// TIA Portal V16 export
// export: Created 2021-08-10T09:04:59.4784454Z, ExportSetting WithDefaults, WithReadOnly, DisplayName Totally Integrated Automation Portal, DisplayVersion V16, DisplayName TIA Portal Version Control Interface, DisplayVersion V16, DisplayName TIA Portal Openness, DisplayVersion V16, DisplayName TIA Portal Teamcenter Gateway, DisplayVersion V16, DisplayName SINAMICS Startdrive Advanced, DisplayVersion V16, DisplayName SINAMICS Startdrive G130, G150, S120, S150, SINAMICS MV, S210, DisplayVersion V16, DisplayName SINAMICS Startdrive G110M, G120, G120C, G120D, G120P, DisplayVersion V16, DisplayName STEP 7 Professional, DisplayVersion V16, DisplayName STEP 7 Safety, DisplayVersion V16, DisplayName WinCC Unified SCADA Engineering System, DisplayVersion V16
FUNCTION_BLOCK "Valve Liquid 2"   // FB3, FBD
{ S7_Optimized_Access := 'TRUE' }
VERSION : 0.1
// stored: AutoNumber true, CodeModifiedDate 2020-02-26T13:09:02.1361563Z, CompileDate 2021-07-03T08:38:43.4120873Z, CreationDate 2020-02-26T07:16:44.3135253Z, DownloadWithoutReinit false, HandleErrorsWithinBlock false, InterfaceModifiedDate 2020-02-26T12:49:56.0619358Z, IsConsistent true, IsIECCheckEnabled false, IsKnowHowProtected false, ISMultiInstanceCapable true, IsRetainMemResEnabled false, IsWriteProtected false, LibraryConformanceStatus Warning: The object contains access to global data blocks. Warning: The block contains direct access to inputs, outputs, bit memories, indirect access to the registry or indirect access to external memory areas that are unknown at the time of compilation., MemoryReserve 100, ModifiedDate 2020-02-26T13:09:02.1361563Z, ParameterModified 2020-02-26T07:16:44.3135253Z, PLCSimAdvancedSupport true, SetENOAutomatically false, StructureModified 2020-02-26T12:49:56.0619358Z, UDAEnableTagReadback false
   VAR
      VlvLiq2 : "fbValve_Solenoid";
   END_VAR
BEGIN

REGION Network 1
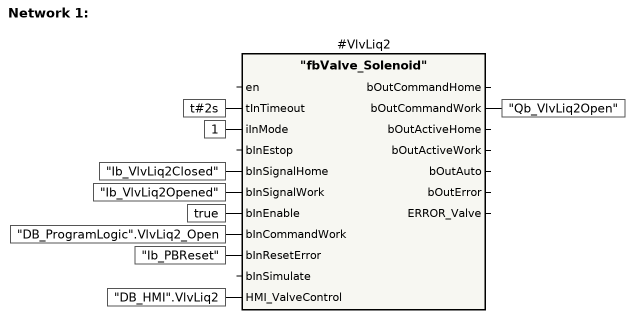
   #VlvLiq2(tInTimeout := t#2s,   // "fbValve_Solenoid"
            iInMode := 1,
            bInSignalHome := "Ib_VlvLiq2Closed",
            bInSignalWork := "Ib_VlvLiq2Opened",
            bInEnable := true,
            bInCommandWork := "DB_ProgramLogic".VlvLiq2_Open,
            bInResetError := "Ib_PBReset",
            HMI_ValveControl := "DB_HMI".VlvLiq2,
            bOutCommandWork => "Qb_VlvLiq2Open");
END_REGION
END_FUNCTION_BLOCK
